FUNCTION_BLOCK FB_GPI_Test EXTENDS TcUnit.FB_TestSuite
VAR_INPUT
END_VAR
VAR_OUTPUT
END_VAR
VAR
    fb_MKS275: FB_MKS275;
    fb_MKS317: FB_MKS317;
    i_iPRESS_R AT %Q* :INT;
    cycle:INT :=0;
END_VAR

M_INIT();
M_CheckRange();
cycle:=cycle+1;

METHOD M_CheckRange
VAR
    Expected:REAL;
    Actual:REAL;
    eStateExpected: E_PressureState;
    eStateActual: E_PressureState;
END_VAR

TEST('MKS275_Check_Range');
Case cycle of
    4:
    This^.i_iPRESS_R := V_TO_INT(3.674);
    Expected :=5 ;
    eStateExpected := Valid;

    7:
    TEST('MKS275_Range_R2');
    Actual := This^.fb_MKS275.PG.rPRESS;
    eStateActual := This^.fb_MKS275.PG.eState;
    AssertTrue(This^.fb_MKS275.PG.xPRESS_OK, 'MKS275 xPRESS_OK is set to False');
    AssertEquals(eStateExpected,eStateActual,'MKS275 eState Fail');
    AssertEquals_REAL(Expected, Actual,0.1, 'MKS275 rPress Fail');
    TEST_FINISHED_NAMED('MKS275_Range_R2');

    8:
    This^.i_iPRESS_R := V_TO_INT(5.614);
    Expected :=900 ;
    eStateExpected := Valid;


    12:
    TEST('MKS275_Range_R3');
    Actual := This^.fb_MKS275.PG.rPRESS;
    eStateActual := This^.fb_MKS275.PG.eState;
    AssertTrue(This^.fb_MKS275.PG.xPRESS_OK, 'MKS275 xPRESS_OK is set to False');
    AssertEquals(eStateExpected,eStateActual,'MKS275 eState Fail');
    AssertEquals_REAL(Expected, Actual,1, 'MKS275 rPress Fail');
    TEST_FINISHED_NAMED('MKS275_Range_R3');


    13:
    This^.i_iPRESS_R := V_TO_INT(0.3);
    Expected :=-1 ;
    eStateExpected := GaugeDisconnected;

    17:
    TEST('MKS275_Range_Off');
    Actual := This^.fb_MKS275.PG.rPRESS;
    eStateActual := This^.fb_MKS275.PG.eState;
    AssertTrue(This^.fb_MKS275.PG.xPRESS_OK, 'MKS275 xPRESS_OK is set to False');
    AssertEquals(eStateExpected,eStateActual,'MKS275 eState Fail');
    AssertEquals_REAL(Expected, Actual,1, 'MKS275 rPress Fail');
    TEST_FINISHED_NAMED('MKS275_Range_Off');


    18:
    This^.i_iPRESS_R := V_TO_INT(5.66);
    Expected :=-1 ;
    eStateExpected := OoR;

    22:
    TEST('MKS275_Range_OoR');
    Actual := This^.fb_MKS275.PG.rPRESS;
    eStateActual := This^.fb_MKS275.PG.eState;
    AssertTrue(This^.fb_MKS275.PG.xPRESS_OK, 'MKS275 xPRESS_OK is set to False');
    AssertEquals(eStateExpected,eStateActual,'MKS275 eState Fail');
    AssertEquals_REAL(Expected, Actual,1, 'MKS275 rPress Fail');
    TEST_FINISHED_NAMED('MKS275_Range_OoR');
    TEST_FINISHED_NAMED('MKS275_Check_Range');

END_CASE

This^.fb_MKS275(PG=>);
This^.fb_MKS317(PG=>);
END_METHOD

METHOD M_INIT
VAR
    Expected:REAL;
    Actual:REAL;
    eStateExpected: E_PressureState;
    eStateActual: E_PressureState;
END_VAR
// Start the Test
TEST('MKS275_Startup');
//Assign Voltage to FB
This^.i_iPRESS_R := V_TO_INT(0.384);
// Assigne expected result corresponing to the test input
Expected :=0.001 ;
eStateExpected := Valid;
//Instantiate the function block
This^.fb_MKS275(PG=>);
// Wait for few cycles
IF( cycle = 3) THEN
    // Check the results
    Actual := This^.fb_MKS275.PG.rPRESS;
    eStateActual := This^.fb_MKS275.PG.eState;
    AssertTrue(This^.fb_MKS275.PG.xPRESS_OK, 'MKS275 xPRESS_OK is set to False');
    AssertEquals(eStateExpected,eStateActual,'MKS275 eState Fail');
    AssertEquals_REAL(Expected, Actual,0.0001, 'MKS275 rPress Fail');
    TEST_FINISHED_NAMED('MKS275_Startup');
END_IF
END_METHOD

END_FUNCTION_BLOCK

(* stored: Version 1.1.0.1
   POU FB_GPI_Test: Id {22be8154-9d2d-4e8a-bd0c-5b5a056f6bed}, SpecialFunc None
   Method M_CheckRange: Id {f9925fbb-0a4e-4266-90b0-bed226f828a8}
   Method M_INIT: Id {e96acaf5-8f1a-41ed-9baa-3496cc1ec916} *)
